FUNCTION_BLOCK Ramp
VAR_INPUT
END_VAR
VAR_OUTPUT
	m_presenceSensorRampFull : PresenceSensor;
END_VAR
VAR
END_VAR

END_FUNCTION_BLOCK

(* stored: Version 1.1.0.1
   POU Ramp: Id {21bef6a5-6483-4a1b-8c60-9287ddbeb696}, SpecialFunc None *)
